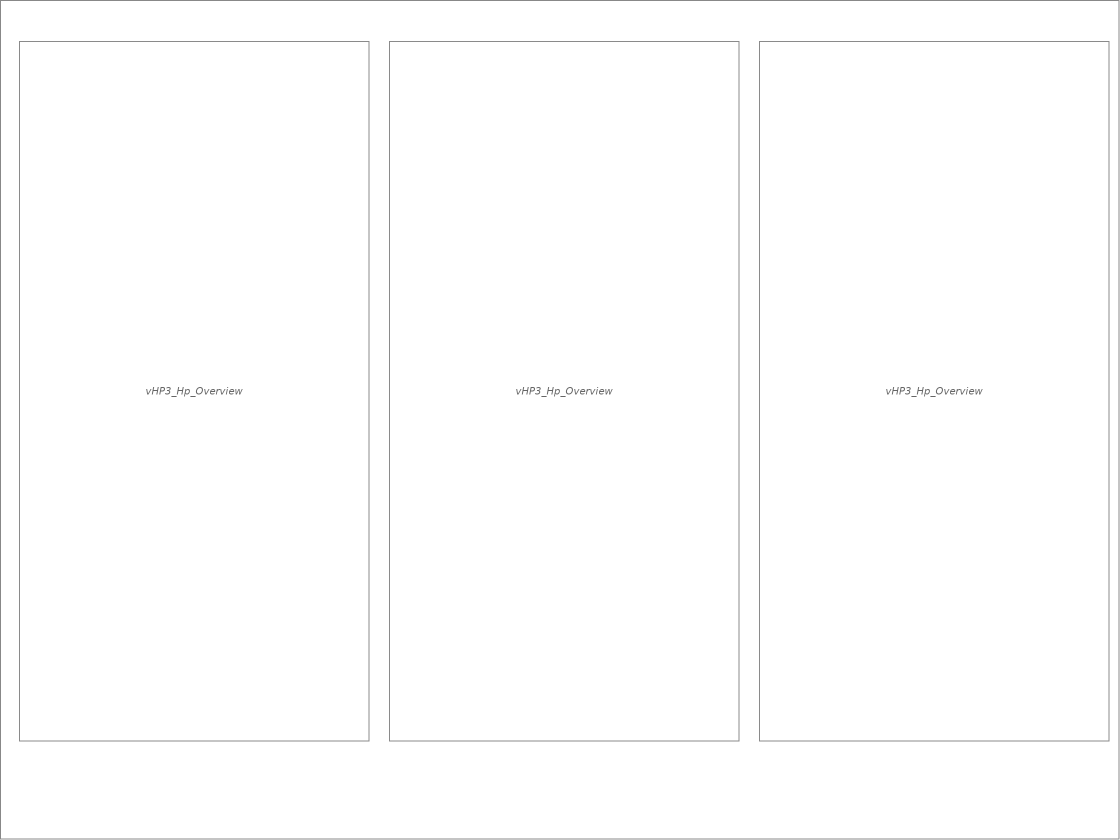
VISUALIZATION vHP3_MachineOverview  // 1120x840
VAR_IN_OUT
	fbHP_M1: fbHPv3_Control;
	fbHP_M2: fbHPv3_Control;
	fbHP_M3: fbHPv3_Control;
END_VAR
    Frame (19,41 350x700)
        shows vHP3_Hp_Overview(fbHP := fbHP_M1)
    Frame (389,41 350x700)
        shows vHP3_Hp_Overview(fbHP := fbHP_M2)
    Frame (759,41 350x700)
        shows vHP3_Hp_Overview(fbHP := fbHP_M3)
END_VISUALIZATION

(* stored: Version 1.1.0.1, ProductVersion 3.1.4024.12
   Visu vHP3_MachineOverview: Id {e4e3d4c5-9515-4ead-a9fb-1f3ab14c0155} *)
